Fanuc KAREL source: NC0088.KL

-- PROVISIONAL review KL for V1013-1; original PC SHA256 4695a19042c558b8a3da2e6e73a88cd22c33c63ec35a87461627665ea6b3cfb9
-- Incomplete behavior may be omitted. Consult companion uncertainty JSON. Do not deploy.
PROGRAM NC0088
%NOLOCKGROUP
-- UNRESOLVED_LOCAL_POOL 4 cells at code offset 3; source declarations unknown
-- DIRECT_LOCAL_WORD_ACCESS alone does not prove INTEGER, REAL, or BOOLEAN
BEGIN
  -- UNRESOLVED_PC offsets 0-8; opcodes 2B,2C,7B
  -- UNRESOLVED_PC offsets 13-20; opcodes 9D,23
  -- UNRESOLVED_PC offsets 25-38; opcodes 21,9D,57,79
  -- UNRESOLVED_PC offsets 43-60; opcodes 21,40,41,42
  -- UNRESOLVED_PC offsets 65-94; opcodes 9D,23,9E,2E,22,7A
  -- UNRESOLVED_PC offsets 99-116; opcodes 21,2E,59,79
  -- UNRESOLVED_PC offsets 121-134; opcodes 21,9D,57,79
  -- UNRESOLVED_PC offsets 139-156; opcodes 21,40,41,42
  -- UNRESOLVED_PC offsets 161-190; opcodes 9D,23,9E,2E,22,7A
  -- UNRESOLVED_PC offsets 195-212; opcodes 21,2E,59,79
  -- UNRESOLVED_PC offsets 217-230; opcodes 21,9D,57,79
  -- UNRESOLVED_PC offsets 235-252; opcodes 21,40,41,42
  -- UNRESOLVED_PC offsets 257-286; opcodes 9D,23,9E,2E,22,7A
  -- UNRESOLVED_PC offsets 291-308; opcodes 21,2E,59,79
  -- UNRESOLVED_PC offsets 313-327; opcodes 21,9D,52,23
  -- UNRESOLVED_PC offsets 332-337; opcodes 7A
  -- UNRESOLVED_PC offsets 342-373; opcodes 20,2C,23,7A,40,41,42
  -- UNRESOLVED_PC offsets 378-402; opcodes 21,2E,52,23,7A,43
  -- UNRESOLVED_PC offsets 407-425; opcodes 21,2E,52,23
  -- UNRESOLVED_PC offsets 435-440; opcodes 7A
  -- UNRESOLVED_PC offsets 445-463; opcodes 21,2E,52,23
  -- UNRESOLVED_PC offsets 473-478; opcodes 7A
  -- UNRESOLVED_PC offsets 483-514; opcodes 20,2C,23,7A,40,41,42
  -- UNRESOLVED_PC offsets 519-543; opcodes 21,2E,52,23,7A,43
  -- UNRESOLVED_PC offsets 548-566; opcodes 21,2E,52,23
  -- UNRESOLVED_PC offsets 576-581; opcodes 7A
  -- UNRESOLVED_PC offsets 586-604; opcodes 21,2E,52,23
  -- UNRESOLVED_PC offsets 614-619; opcodes 7A
  -- UNRESOLVED_PC offsets 624-655; opcodes 20,2C,23,7A,40,41,42
  -- UNRESOLVED_PC offsets 660-684; opcodes 21,2E,52,23,7A,43
  -- UNRESOLVED_PC offsets 689-707; opcodes 21,2E,52,23
  -- UNRESOLVED_PC offsets 717-722; opcodes 7A
  -- UNRESOLVED_PC offsets 727-745; opcodes 21,2E,52,23
  -- UNRESOLVED_PC offsets 755-759; opcodes 7F
  -- UNRESOLVED_PC offsets 764-768; opcodes 27,AA
  -- UNRESOLVED_PC offsets 773-777; opcodes 7F
END NC0088
